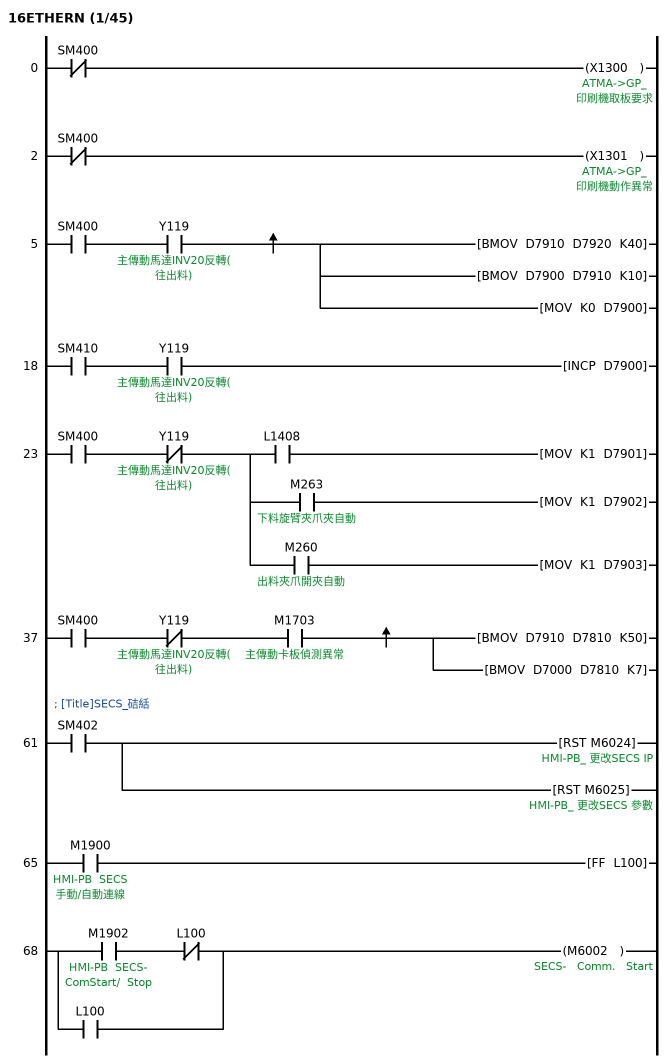
[picture p96: ladder of 16ETHERN, rungs at steps 0 to 68]
0     LDI     SM400
      OUT     X1300  ; ATMA->GP_印刷機取板要求
2     LDI     SM400
      OUT     X1301  ; ATMA->GP_印刷機動作異常
5     LD      SM400
      AND     Y119  ; 主傳動馬達INV20反轉(往出料)
      MEP
      BMOV    D7910 D7920 K40
      BMOV    D7900 D7910 K10
      MOV     K0 D7900
18    LD      SM410
      AND     Y119  ; 主傳動馬達INV20反轉(往出料)
      INCP    D7900
23    LD      SM400
      ANI     Y119  ; 主傳動馬達INV20反轉(往出料)
      MPS
      AND     L1408
      MOV     K1 D7901
      MRD
      AND     M263  ; 下料旋臂夾爪夾自動
      MOV     K1 D7902
      MPP
      AND     M260  ; 出料夾爪開夾自動
      MOV     K1 D7903
37    LD      SM400
      ANI     Y119  ; 主傳動馬達INV20反轉(往出料)
      AND     M1703  ; 主傳動卡板偵測異常
      MEP
      BMOV    D7910 D7810 K50
      BMOV    D7000 D7810 K7
; [Title]SECS_連線
61    LD      SM402
      RST     M6024  ; HMI-PB_ 更改SECS IP
      RST     M6025  ; HMI-PB_ 更改SECS 參數
65    LD      M1900  ; HMI-PB  SECS    手動/自動連線
      FF      L100
68    LD      M1902  ; HMI-PB  SECS-ComStart/  Stop
      ANI     L100
      OR      L100
      OUT     M6002  ; SECS-   Comm.   Start
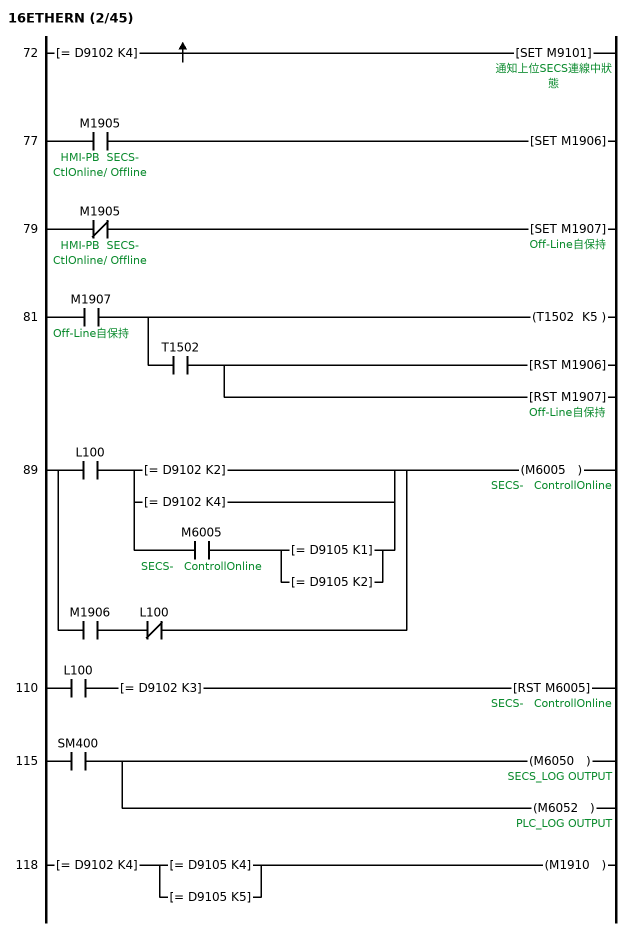
72    LD=     D9102 K4
      MEP
      SET     M9101  ; 通知上位SECS連線中狀態
77    LD      M1905  ; HMI-PB  SECS-CtlOnline/ Offline
      SET     M1906
79    LDI     M1905  ; HMI-PB  SECS-CtlOnline/ Offline
      SET     M1907  ; Off-Line自保持
81    LD      M1907  ; Off-Line自保持
      OUT     T1502 K5
      AND     T1502
      RST     M1906
      RST     M1907  ; Off-Line自保持
89    LD      L100
      LD=     D9102 K2
      OR=     D9102 K4
      LD      M6005  ; SECS-   ControllOnline
      LD=     D9105 K1
      OR=     D9105 K2
      ANB
      ORB
      ANB
      LD      M1906
      ANI     L100
      ORB
      OUT     M6005  ; SECS-   ControllOnline
110   LD      L100
      AND=    D9102 K3
      RST     M6005  ; SECS-   ControllOnline
115   LD      SM400
      OUT     M6050  ; SECS_LOG OUTPUT
      OUT     M6052  ; PLC_LOG OUTPUT
118   LD=     D9102 K4
      LD=     D9105 K4
      OR=     D9105 K5
      ANB
      OUT     M1910
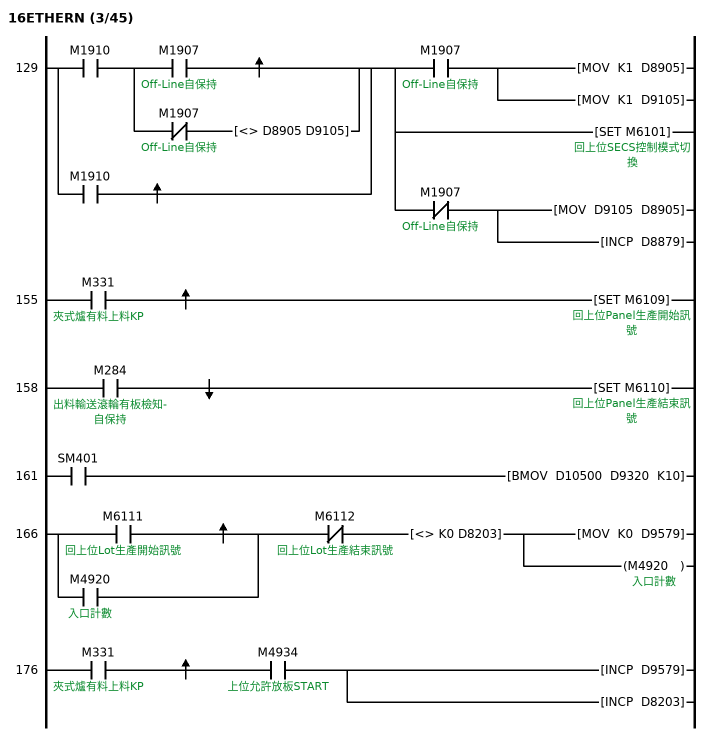
129   LD      M1910
      LD      M1907  ; Off-Line自保持
      MEP
      LDI     M1907  ; Off-Line自保持
      AND<>   D8905 D9105
      ORB
      ANB
      LD      M1910
      MEP
      ORB
      MPS
      AND     M1907  ; Off-Line自保持
      MOV     K1 D8905
      MOV     K1 D9105
      MPP
      SET     M6101  ; 回上位SECS控制模式切換
      ANI     M1907  ; Off-Line自保持
      MOV     D9105 D8905
      INCP    D8879
155   LD      M331  ; 夾式爐有料上料KP
      MEP
      SET     M6109  ; 回上位Panel生產開始訊號
158   LD      M284  ; 出料輸送滾輪有板檢知-自保持
      MEF
      SET     M6110  ; 回上位Panel生產結束訊號
161   LD      SM401
      BMOV    D10500 D9320 K10
166   LD      M6111  ; 回上位Lot生產開始訊號
      MEP
      OR      M4920  ; 入口計數
      ANI     M6112  ; 回上位Lot生產結束訊號
      AND<>   K0 D8203
      MOV     K0 D9579
      OUT     M4920  ; 入口計數
176   LD      M331  ; 夾式爐有料上料KP
      MEP
      AND     M4934  ; 上位允許放板START
      INCP    D9579
      INCP    D8203
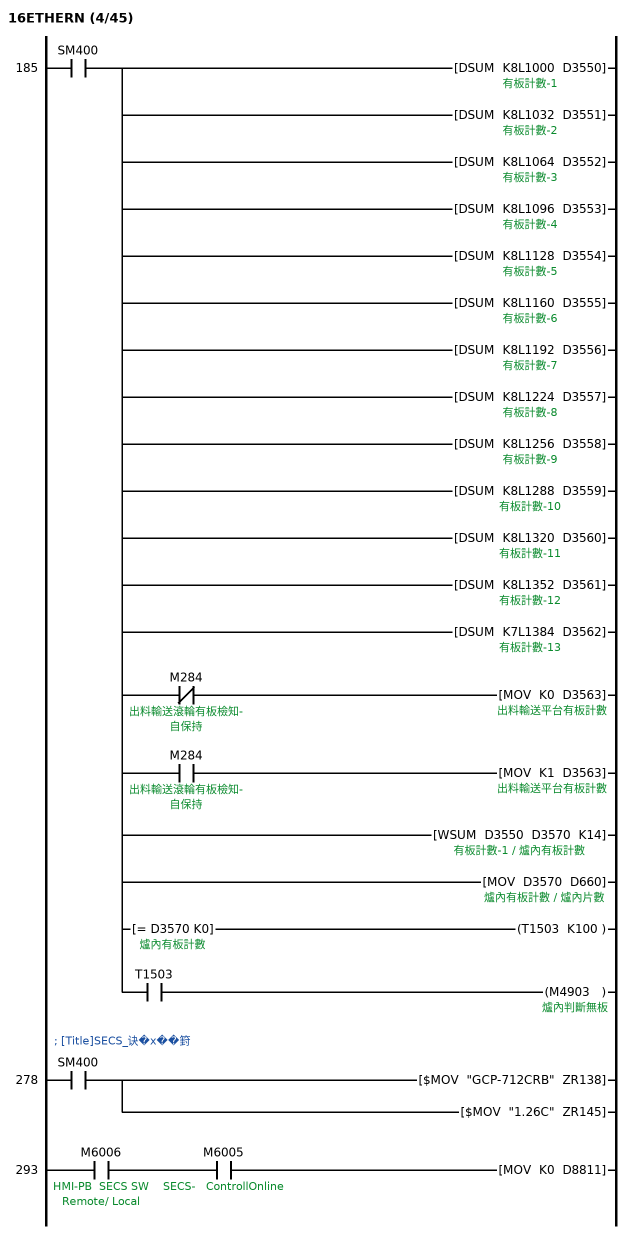
185   LD      SM400
      DSUM    K8L1000 D3550  ; 有板計數-1
      DSUM    K8L1032 D3551  ; 有板計數-2
      DSUM    K8L1064 D3552  ; 有板計數-3
      DSUM    K8L1096 D3553  ; 有板計數-4
      DSUM    K8L1128 D3554  ; 有板計數-5
      DSUM    K8L1160 D3555  ; 有板計數-6
      DSUM    K8L1192 D3556  ; 有板計數-7
      DSUM    K8L1224 D3557  ; 有板計數-8
      DSUM    K8L1256 D3558  ; 有板計數-9
      DSUM    K8L1288 D3559  ; 有板計數-10
      DSUM    K8L1320 D3560  ; 有板計數-11
      DSUM    K8L1352 D3561  ; 有板計數-12
      DSUM    K7L1384 D3562  ; 有板計數-13
      MPS
      ANI     M284  ; 出料輸送滾輪有板檢知-自保持
      MOV     K0 D3563  ; 出料輸送平台有板計數
      MRD
      AND     M284  ; 出料輸送滾輪有板檢知-自保持
      MOV     K1 D3563
      MPP
      WSUM    D3550 D3570 K14  ; 爐內有板計數
      MOV     D3570 D660  ; 爐內片數
      MPS
      AND=    D3570 K0  ; 爐內有板計數
      OUT     T1503 K100
      MPP
      AND     T1503
      OUT     M4903  ; 爐內判斷無板
; [Title]SECS_機台狀態
278   LD      SM400
      $MOV    "GCP-712CRB" ZR138
      $MOV    "1.26C" ZR145
293   LD      M6006  ; HMI-PB  SECS SW  Remote/ Local
      AND     M6005  ; SECS-   ControllOnline
      MOV     K0 D8811
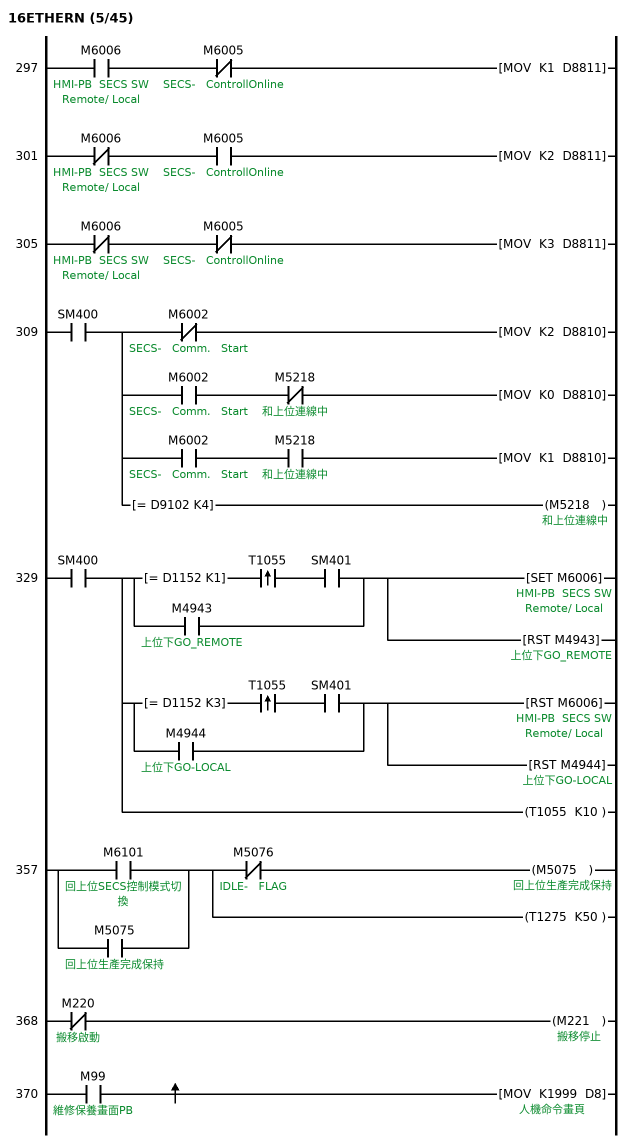
297   LD      M6006  ; HMI-PB  SECS SW  Remote/ Local
      ANI     M6005  ; SECS-   ControllOnline
      MOV     K1 D8811
301   LDI     M6006  ; HMI-PB  SECS SW  Remote/ Local
      AND     M6005  ; SECS-   ControllOnline
      MOV     K2 D8811
305   LDI     M6006  ; HMI-PB  SECS SW  Remote/ Local
      ANI     M6005  ; SECS-   ControllOnline
      MOV     K3 D8811
309   LD      SM400
      MPS
      ANI     M6002  ; SECS-   Comm.   Start
      MOV     K2 D8810
      MRD
      AND     M6002  ; SECS-   Comm.   Start
      ANI     M5218  ; 和上位連線中
      MOV     K0 D8810
      MRD
      AND     M6002  ; SECS-   Comm.   Start
      AND     M5218  ; 和上位連線中
      MOV     K1 D8810
      MPP
      AND=    D9102 K4
      OUT     M5218  ; 和上位連線中
329   LD      SM400
      MPS
      LD=     D1152 K1
      ANDP    T1055
      AND     SM401
      OR      M4943  ; 上位下GO_REMOTE
      ANB
      SET     M6006  ; HMI-PB  SECS SW  Remote/ Local
      RST     M4943  ; 上位下GO_REMOTE
      MRD
      LD=     D1152 K3
      ANDP    T1055
      AND     SM401
      OR      M4944  ; 上位下GO-LOCAL
      ANB
      RST     M6006  ; HMI-PB  SECS SW  Remote/ Local
      RST     M4944  ; 上位下GO-LOCAL
      MPP
      OUT     T1055 K10
357   LD      M6101  ; 回上位SECS控制模式切換
      OR      M5075  ; 回上位生產完成保持
      MPS
      ANI     M5076  ; IDLE-   FLAG
      OUT     M5075  ; 回上位生產完成保持
      MPP
      OUT     T1275 K50
368   LDI     M220  ; 搬移啟動
      OUT     M221  ; 搬移停止
370   LD      M99  ; 維修保養畫面PB
      MEP
      MOV     K1999 D8  ; 人機命令畫頁
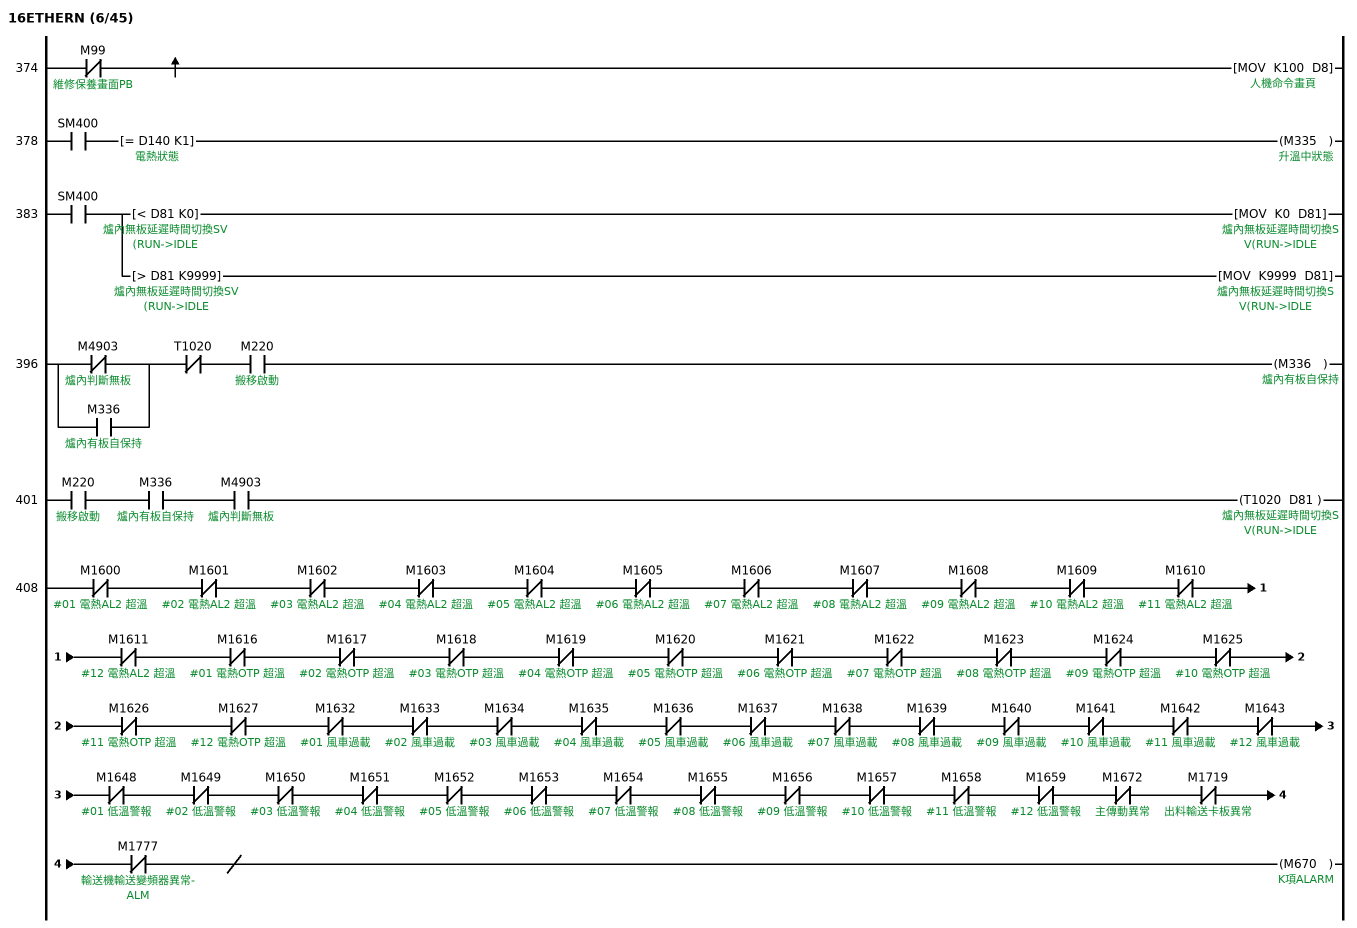
374   LDI     M99  ; 維修保養畫面PB
      MEP
      MOV     K100 D8
378   LD      SM400
      AND=    D140 K1  ; 電熱狀態
      OUT     M335  ; 升溫中狀態
383   LD      SM400
      MPS
      AND<    D81 K0  ; 爐內無板延遲時間切換SV(RUN->IDLE
      MOV     K0 D81
      MPP
      AND>    D81 K9999  ; 爐內無板延遲時間切換SV(RUN->IDLE
      MOV     K9999 D81
396   LDI     M4903  ; 爐內判斷無板
      OR      M336  ; 爐內有板自保持
      ANI     T1020
      AND     M220  ; 搬移啟動
      OUT     M336  ; 爐內有板自保持
401   LD      M220  ; 搬移啟動
      AND     M336  ; 爐內有板自保持
      AND     M4903  ; 爐內判斷無板
      OUT     T1020 D81  ; 爐內無板延遲時間切換SV(RUN->IDLE
408   LDI     M1600  ; #01 電熱AL2 超溫
      ANI     M1601  ; #02 電熱AL2 超溫
      ANI     M1602  ; #03 電熱AL2 超溫
      ANI     M1603  ; #04 電熱AL2 超溫
      ANI     M1604  ; #05 電熱AL2 超溫
      ANI     M1605  ; #06 電熱AL2 超溫
      ANI     M1606  ; #07 電熱AL2 超溫
      ANI     M1607  ; #08 電熱AL2 超溫
      ANI     M1608  ; #09 電熱AL2 超溫
      ANI     M1609  ; #10 電熱AL2 超溫
      ANI     M1610  ; #11 電熱AL2 超溫
      ANI     M1611  ; #12 電熱AL2 超溫
      ANI     M1616  ; #01 電熱OTP 超溫
      ANI     M1617  ; #02 電熱OTP 超溫
      ANI     M1618  ; #03 電熱OTP 超溫
      ANI     M1619  ; #04 電熱OTP 超溫
      ANI     M1620  ; #05 電熱OTP 超溫
      ANI     M1621  ; #06 電熱OTP 超溫
      ANI     M1622  ; #07 電熱OTP 超溫
      ANI     M1623  ; #08 電熱OTP 超溫
      ANI     M1624  ; #09 電熱OTP 超溫
      ANI     M1625  ; #10 電熱OTP 超溫
      ANI     M1626  ; #11 電熱OTP 超溫
      ANI     M1627  ; #12 電熱OTP 超溫
      ANI     M1632  ; #01 風車過載
      ANI     M1633  ; #02 風車過載
      ANI     M1634  ; #03 風車過載
      ANI     M1635  ; #04 風車過載
      ANI     M1636  ; #05 風車過載
      ANI     M1637  ; #06 風車過載
      ANI     M1638  ; #07 風車過載
      ANI     M1639  ; #08 風車過載
      ANI     M1640  ; #09 風車過載
      ANI     M1641  ; #10 風車過載
      ANI     M1642  ; #11 風車過載
      ANI     M1643  ; #12 風車過載
      ANI     M1648  ; #01 低溫警報
      ANI     M1649  ; #02 低溫警報
      ANI     M1650  ; #03 低溫警報
      ANI     M1651  ; #04 低溫警報
      ANI     M1652  ; #05 低溫警報
      ANI     M1653  ; #06 低溫警報
      ANI     M1654  ; #07 低溫警報
      ANI     M1655  ; #08 低溫警報
      ANI     M1656  ; #09 低溫警報
      ANI     M1657  ; #10 低溫警報
      ANI     M1658  ; #11 低溫警報
      ANI     M1659  ; #12 低溫警報
      ANI     M1672  ; 主傳動異常
      ANI     M1719  ; 出料輸送卡板異常
      ANI     M1777  ; 輸送機輸送變頻器異常-ALM
      INV
      OUT     M670  ; K項ALARM
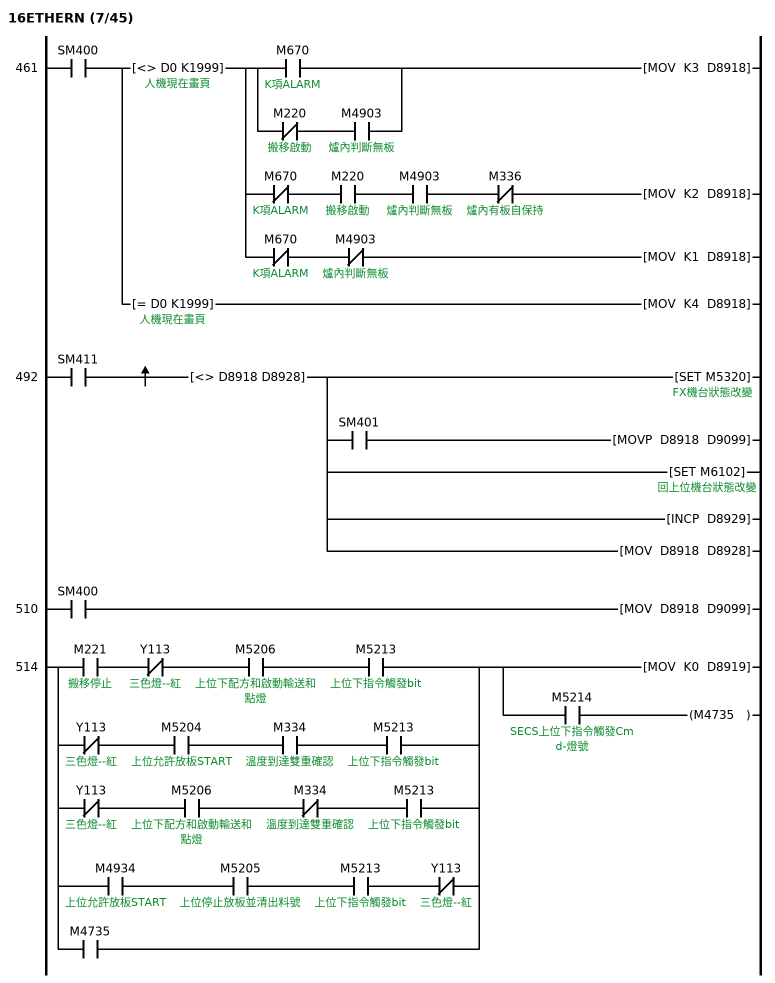
461   LD      SM400
      MPS
      AND<>   D0 K1999  ; 人機現在畫頁
      MPS
      LD      M670  ; K項ALARM
      LDI     M220  ; 搬移啟動
      AND     M4903  ; 爐內判斷無板
      ORB
      ANB
      MOV     K3 D8918
      MRD
      ANI     M670  ; K項ALARM
      AND     M220  ; 搬移啟動
      AND     M4903  ; 爐內判斷無板
      ANI     M336  ; 爐內有板自保持
      MOV     K2 D8918
      MPP
      ANI     M670  ; K項ALARM
      ANI     M4903  ; 爐內判斷無板
      MOV     K1 D8918
      MPP
      AND=    D0 K1999  ; 人機現在畫頁
      MOV     K4 D8918
492   LD      SM411
      MEP
      AND<>   D8918 D8928
      SET     M5320  ; FX機台狀態改變
      MPS
      AND     SM401
      MOVP    D8918 D9099
      MPP
      SET     M6102  ; 回上位機台狀態改變
      INCP    D8929
      MOV     D8918 D8928
510   LD      SM400
      MOV     D8918 D9099
514   LD      M221  ; 搬移停止
      ANI     Y113  ; 三色燈--紅
      AND     M5206  ; 上位下配方和啟動輸送和點燈
      AND     M5213  ; 上位下指令觸發bit
      LDI     Y113  ; 三色燈--紅
      AND     M5204  ; 上位允許放板START
      AND     M334  ; 溫度到達雙重確認
      AND     M5213  ; 上位下指令觸發bit
      ORB
      LDI     Y113  ; 三色燈--紅
      AND     M5206  ; 上位下配方和啟動輸送和點燈
      ANI     M334  ; 溫度到達雙重確認
      AND     M5213  ; 上位下指令觸發bit
      ORB
      LD      M4934  ; 上位允許放板START
      AND     M5205  ; 上位停止放板並清出料號
      AND     M5213  ; 上位下指令觸發bit
      ANI     Y113  ; 三色燈--紅
      ORB
      OR      M4735
      MOV     K0 D8919
      AND     M5214  ; SECS上位下指令觸發Cmd-燈號
      OUT     M4735
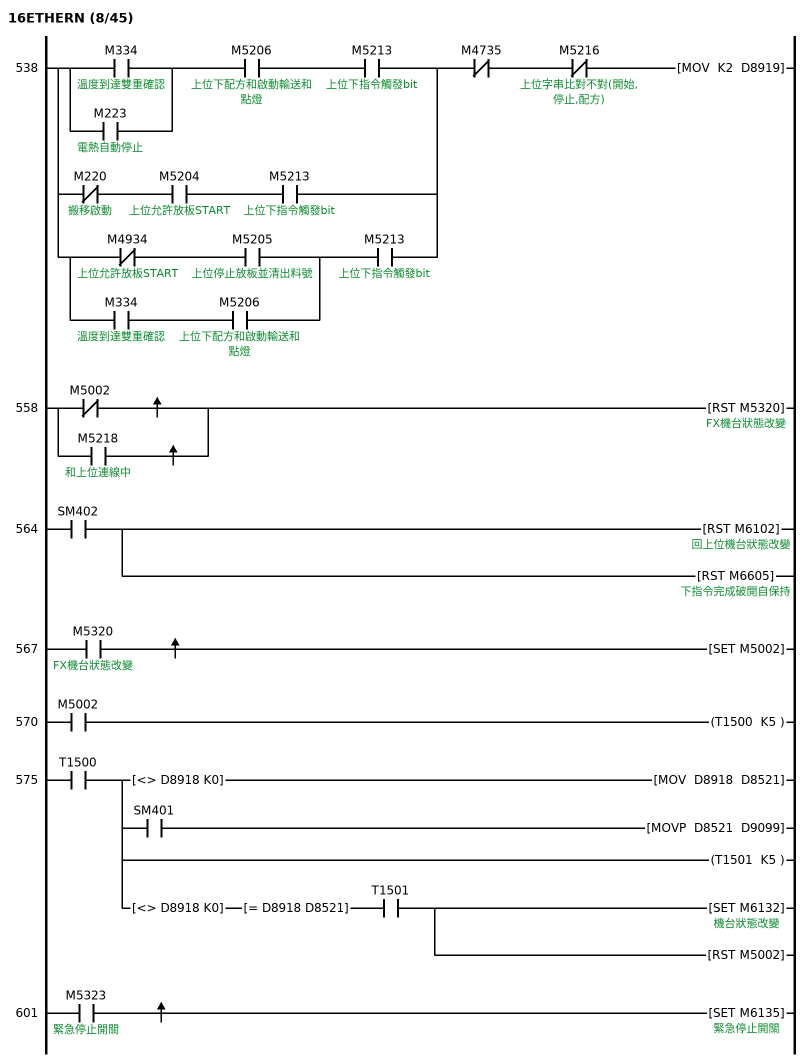
538   LD      M334  ; 溫度到達雙重確認
      OR      M223  ; 電熱自動停止
      AND     M5206  ; 上位下配方和啟動輸送和點燈
      AND     M5213  ; 上位下指令觸發bit
      LDI     M220  ; 搬移啟動
      AND     M5204  ; 上位允許放板START
      AND     M5213  ; 上位下指令觸發bit
      ORB
      LDI     M4934  ; 上位允許放板START
      AND     M5205  ; 上位停止放板並清出料號
      LD      M334  ; 溫度到達雙重確認
      AND     M5206  ; 上位下配方和啟動輸送和點燈
      ORB
      AND     M5213  ; 上位下指令觸發bit
      ORB
      ANI     M4735
      ANI     M5216  ; 上位字串比對不對(開始,停止,配方)
      MOV     K2 D8919
558   LDI     M5002
      MEP
      LD      M5218  ; 和上位連線中
      MEP
      ORB
      RST     M5320  ; FX機台狀態改變
564   LD      SM402
      RST     M6102  ; 回上位機台狀態改變
      RST     M6605  ; 下指令完成破開自保持
567   LD      M5320  ; FX機台狀態改變
      MEP
      SET     M5002
570   LD      M5002
      OUT     T1500 K5
575   LD      T1500
      MPS
      AND<>   D8918 K0
      MOV     D8918 D8521
      MRD
      AND     SM401
      MOVP    D8521 D9099
      MPP
      OUT     T1501 K5
      AND<>   D8918 K0
      AND=    D8918 D8521
      AND     T1501
      SET     M6132  ; 機台狀態改變
      RST     M5002
601   LD      M5323  ; 緊急停止開關
      MEP
      SET     M6135  ; 緊急停止開關
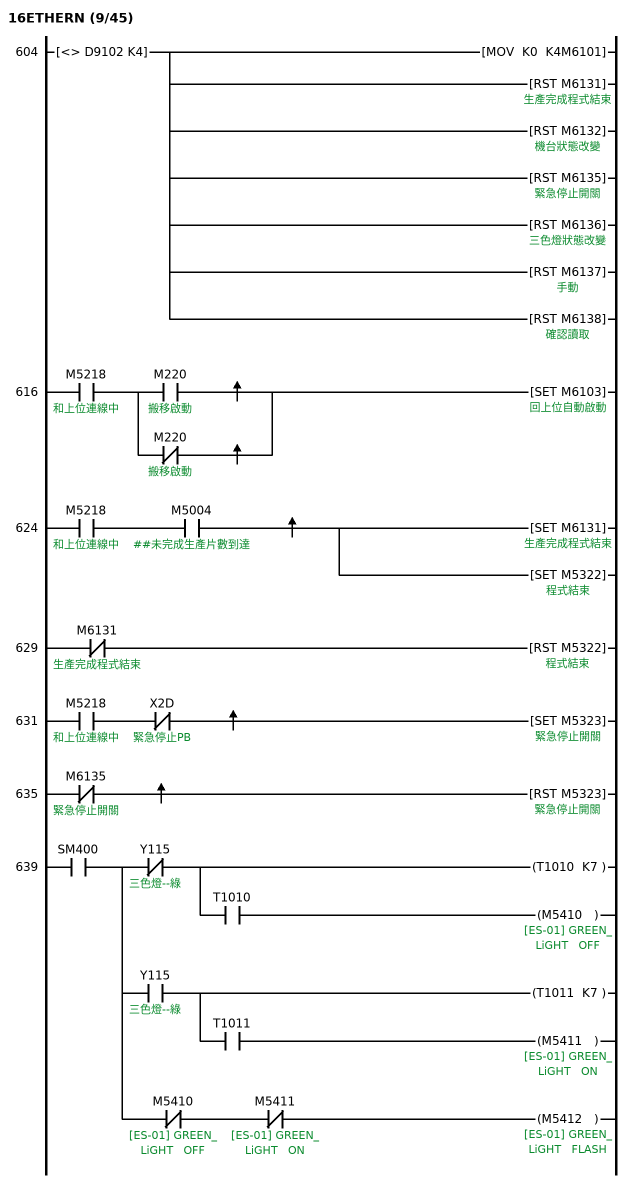
604   LD<>    D9102 K4
      MOV     K0 K4M6101
      RST     M6131  ; 生產完成程式結束
      RST     M6132  ; 機台狀態改變
      RST     M6135  ; 緊急停止開關
      RST     M6136  ; 三色燈狀態改變
      RST     M6137  ; 手動
      RST     M6138  ; 確認讀取
616   LD      M5218  ; 和上位連線中
      LD      M220  ; 搬移啟動
      MEP
      LDI     M220  ; 搬移啟動
      MEP
      ORB
      ANB
      SET     M6103  ; 回上位自動啟動
624   LD      M5218  ; 和上位連線中
      AND     M5004  ; ##未完成生產片數到達
      MEP
      SET     M6131  ; 生產完成程式結束
      SET     M5322  ; 程式結束
629   LDI     M6131  ; 生產完成程式結束
      RST     M5322  ; 程式結束
631   LD      M5218  ; 和上位連線中
      ANI     X2D  ; 緊急停止PB
      MEP
      SET     M5323  ; 緊急停止開關
635   LDI     M6135  ; 緊急停止開關
      MEP
      RST     M5323  ; 緊急停止開關
639   LD      SM400
      MPS
      ANI     Y115  ; 三色燈--綠
      OUT     T1010 K7
      AND     T1010
      OUT     M5410  ; [ES-01] GREEN_  LiGHT   OFF
      MRD
      AND     Y115  ; 三色燈--綠
      OUT     T1011 K7
      AND     T1011
      OUT     M5411  ; [ES-01] GREEN_  LiGHT   ON
      MPP
      ANI     M5410  ; [ES-01] GREEN_  LiGHT   OFF
      ANI     M5411  ; [ES-01] GREEN_  LiGHT   ON
      OUT     M5412  ; [ES-01] GREEN_  LiGHT   FLASH
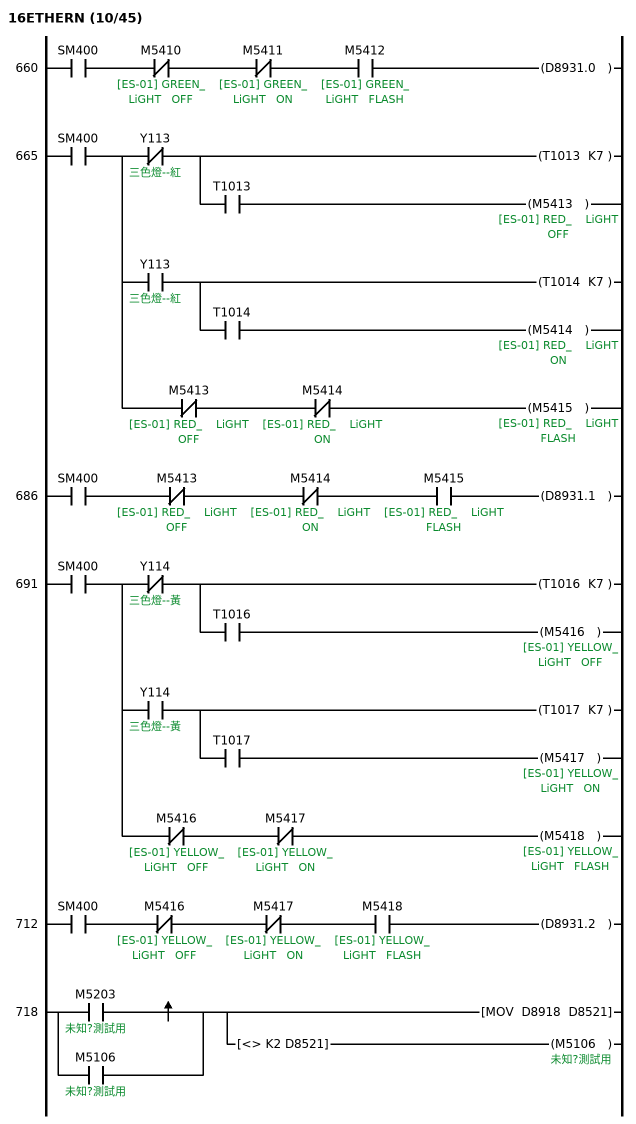
660   LD      SM400
      ANI     M5410  ; [ES-01] GREEN_  LiGHT   OFF
      ANI     M5411  ; [ES-01] GREEN_  LiGHT   ON
      AND     M5412  ; [ES-01] GREEN_  LiGHT   FLASH
      OUT     D8931.0
665   LD      SM400
      MPS
      ANI     Y113  ; 三色燈--紅
      OUT     T1013 K7
      AND     T1013
      OUT     M5413  ; [ES-01] RED_    LiGHT   OFF
      MRD
      AND     Y113  ; 三色燈--紅
      OUT     T1014 K7
      AND     T1014
      OUT     M5414  ; [ES-01] RED_    LiGHT   ON
      MPP
      ANI     M5413  ; [ES-01] RED_    LiGHT   OFF
      ANI     M5414  ; [ES-01] RED_    LiGHT   ON
      OUT     M5415  ; [ES-01] RED_    LiGHT   FLASH
686   LD      SM400
      ANI     M5413  ; [ES-01] RED_    LiGHT   OFF
      ANI     M5414  ; [ES-01] RED_    LiGHT   ON
      AND     M5415  ; [ES-01] RED_    LiGHT   FLASH
      OUT     D8931.1
691   LD      SM400
      MPS
      ANI     Y114  ; 三色燈--黃
      OUT     T1016 K7
      AND     T1016
      OUT     M5416  ; [ES-01] YELLOW_ LiGHT   OFF
      MRD
      AND     Y114  ; 三色燈--黃
      OUT     T1017 K7
      AND     T1017
      OUT     M5417  ; [ES-01] YELLOW_ LiGHT   ON
      MPP
      ANI     M5416  ; [ES-01] YELLOW_ LiGHT   OFF
      ANI     M5417  ; [ES-01] YELLOW_ LiGHT   ON
      OUT     M5418  ; [ES-01] YELLOW_ LiGHT   FLASH
712   LD      SM400
      ANI     M5416  ; [ES-01] YELLOW_ LiGHT   OFF
      ANI     M5417  ; [ES-01] YELLOW_ LiGHT   ON
      AND     M5418  ; [ES-01] YELLOW_ LiGHT   FLASH
      OUT     D8931.2
718   LD      M5203  ; 未知?測試用
      MEP
      OR      M5106  ; 未知?測試用
      MOV     D8918 D8521
      AND<>   K2 D8521
      OUT     M5106  ; 未知?測試用
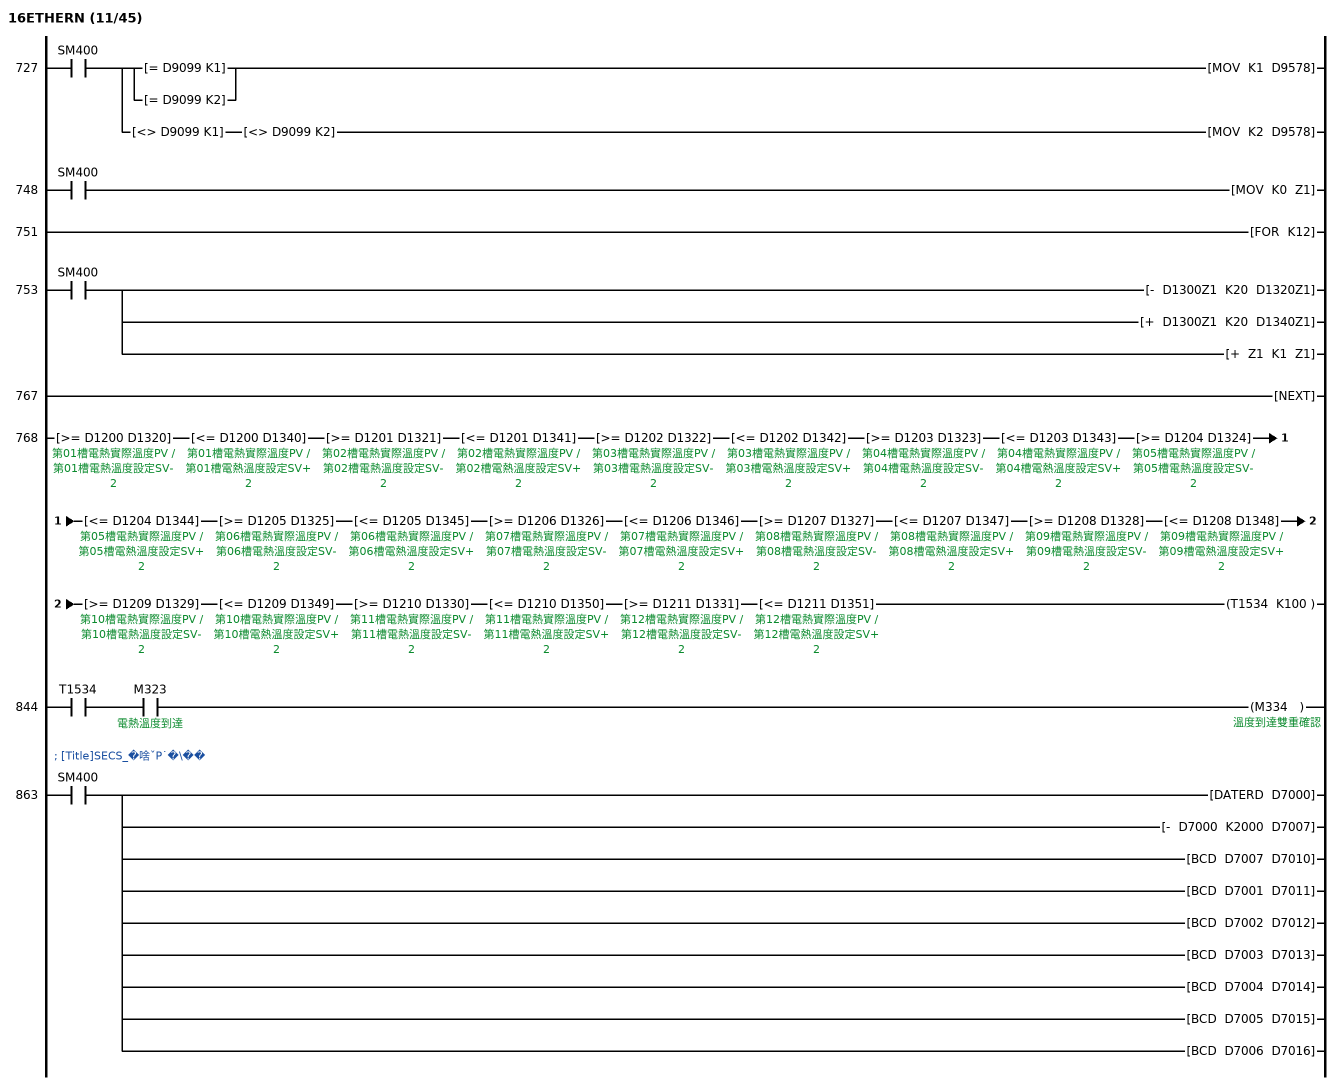
727   LD      SM400
      MPS
      LD=     D9099 K1
      OR=     D9099 K2
      ANB
      MOV     K1 D9578
      MPP
      AND<>   D9099 K1
      AND<>   D9099 K2
      MOV     K2 D9578
748   LD      SM400
      MOV     K0 Z1
751   FOR     K12
753   LD      SM400
      -       D1300Z1 K20 D1320Z1
      +       D1300Z1 K20 D1340Z1
      +       Z1 K1 Z1
767   NEXT
768   LD>=    D1200 D1320  ; 第01槽電熱實際溫度PV / 第01槽電熱溫度設定SV-2
      AND<=   D1200 D1340  ; 第01槽電熱實際溫度PV / 第01槽電熱溫度設定SV+2
      AND>=   D1201 D1321  ; 第02槽電熱實際溫度PV / 第02槽電熱溫度設定SV-2
      AND<=   D1201 D1341  ; 第02槽電熱實際溫度PV / 第02槽電熱溫度設定SV+2
      AND>=   D1202 D1322  ; 第03槽電熱實際溫度PV / 第03槽電熱溫度設定SV-2
      AND<=   D1202 D1342  ; 第03槽電熱實際溫度PV / 第03槽電熱溫度設定SV+2
      AND>=   D1203 D1323  ; 第04槽電熱實際溫度PV / 第04槽電熱溫度設定SV-2
      AND<=   D1203 D1343  ; 第04槽電熱實際溫度PV / 第04槽電熱溫度設定SV+2
      AND>=   D1204 D1324  ; 第05槽電熱實際溫度PV / 第05槽電熱溫度設定SV-2
      AND<=   D1204 D1344  ; 第05槽電熱實際溫度PV / 第05槽電熱溫度設定SV+2
      AND>=   D1205 D1325  ; 第06槽電熱實際溫度PV / 第06槽電熱溫度設定SV-2
      AND<=   D1205 D1345  ; 第06槽電熱實際溫度PV / 第06槽電熱溫度設定SV+2
      AND>=   D1206 D1326  ; 第07槽電熱實際溫度PV / 第07槽電熱溫度設定SV-2
      AND<=   D1206 D1346  ; 第07槽電熱實際溫度PV / 第07槽電熱溫度設定SV+2
      AND>=   D1207 D1327  ; 第08槽電熱實際溫度PV / 第08槽電熱溫度設定SV-2
      AND<=   D1207 D1347  ; 第08槽電熱實際溫度PV / 第08槽電熱溫度設定SV+2
      AND>=   D1208 D1328  ; 第09槽電熱實際溫度PV / 第09槽電熱溫度設定SV-2
      AND<=   D1208 D1348  ; 第09槽電熱實際溫度PV / 第09槽電熱溫度設定SV+2
      AND>=   D1209 D1329  ; 第10槽電熱實際溫度PV / 第10槽電熱溫度設定SV-2
      AND<=   D1209 D1349  ; 第10槽電熱實際溫度PV / 第10槽電熱溫度設定SV+2
      AND>=   D1210 D1330  ; 第11槽電熱實際溫度PV / 第11槽電熱溫度設定SV-2
      AND<=   D1210 D1350  ; 第11槽電熱實際溫度PV / 第11槽電熱溫度設定SV+2
      AND>=   D1211 D1331  ; 第12槽電熱實際溫度PV / 第12槽電熱溫度設定SV-2
      AND<=   D1211 D1351  ; 第12槽電熱實際溫度PV / 第12槽電熱溫度設定SV+2
      OUT     T1534 K100
844   LD      T1534
      AND     M323  ; 電熱溫度到達
      OUT     M334  ; 溫度到達雙重確認
; [Title]SECS_時間同步功能
863   LD      SM400
      DATERD  D7000
      -       D7000 K2000 D7007
      BCD     D7007 D7010
      BCD     D7001 D7011
      BCD     D7002 D7012
      BCD     D7003 D7013
      BCD     D7004 D7014
      BCD     D7005 D7015
      BCD     D7006 D7016
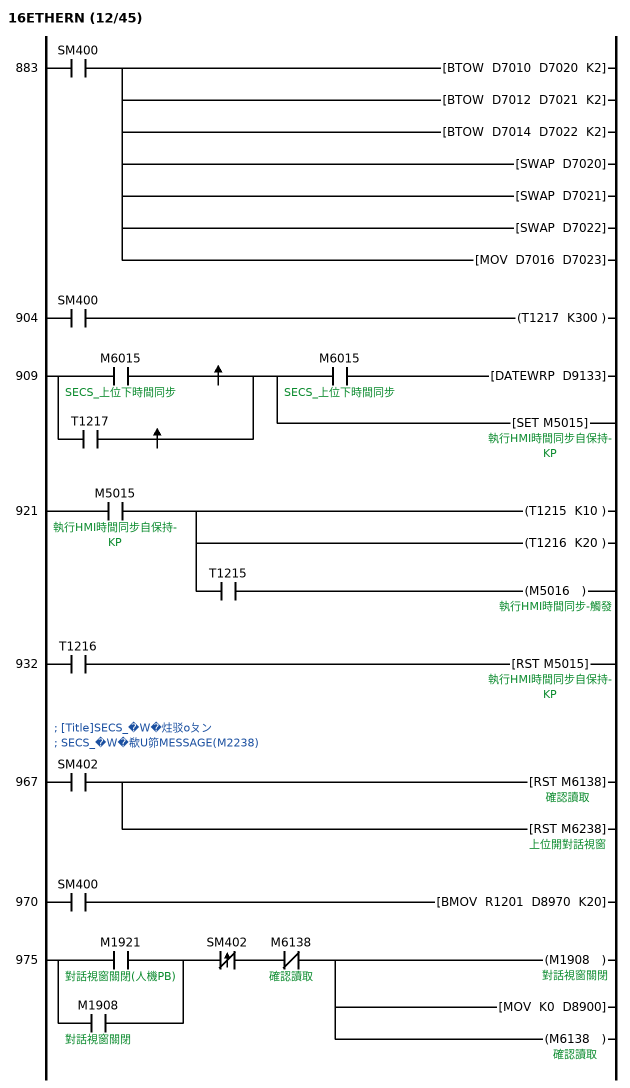
883   LD      SM400
      BTOW    D7010 D7020 K2
      BTOW    D7012 D7021 K2
      BTOW    D7014 D7022 K2
      SWAP    D7020
      SWAP    D7021
      SWAP    D7022
      MOV     D7016 D7023
904   LD      SM400
      OUT     T1217 K300
909   LD      M6015  ; SECS_上位下時間同步
      MEP
      LD      T1217
      MEP
      ORB
      MPS
      AND     M6015  ; SECS_上位下時間同步
      DATEWRP D9133
      MPP
      SET     M5015  ; 執行HMI時間同步自保持-KP
921   LD      M5015  ; 執行HMI時間同步自保持-KP
      OUT     T1215 K10
      OUT     T1216 K20
      AND     T1215
      OUT     M5016  ; 執行HMI時間同步-觸發
932   LD      T1216
      RST     M5015  ; 執行HMI時間同步自保持-KP
; [Title]SECS_上位觸發事件
; SECS_上位下達MESSAGE(M2238)
967   LD      SM402
      RST     M6138  ; 確認讀取
      RST     M6238  ; 上位開對話視窗
970   LD      SM400
      BMOV    R1201 D8970 K20
975   LD      M1921  ; 對話視窗關閉(人機PB)
      OR      M1908  ; 對話視窗關閉
      ANDPI   SM402
      ANI     M6138  ; 確認讀取
      OUT     M1908  ; 對話視窗關閉
      MOV     K0 D8900
      OUT     M6138  ; 確認讀取
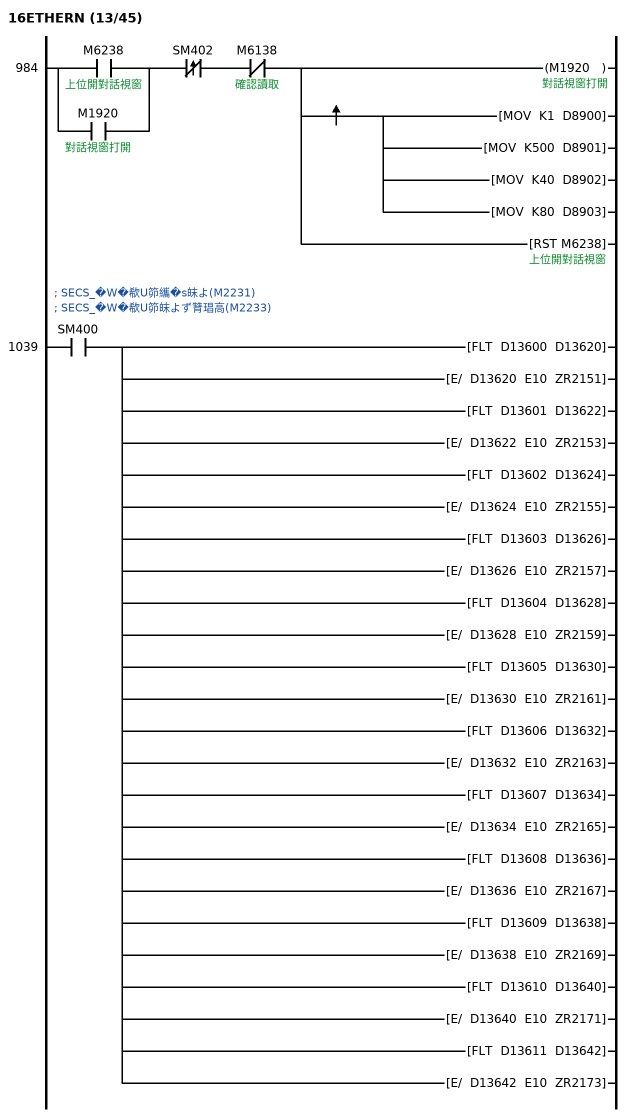
984   LD      M6238  ; 上位開對話視窗
      OR      M1920  ; 對話視窗打開
      ANDPI   SM402
      ANI     M6138  ; 確認讀取
      OUT     M1920  ; 對話視窗打開
      MPS
      MEP
      MOV     K1 D8900
      MOV     K500 D8901
      MOV     K40 D8902
      MOV     K80 D8903
      MPP
      RST     M6238  ; 上位開對話視窗
; SECS_上位下達儲存配方(M2231)
; SECS_上位下達配方內容查詢(M2233)
1039  LD      SM400
      FLT     D13600 D13620
      E/      D13620 E10 ZR2151
      FLT     D13601 D13622
      E/      D13622 E10 ZR2153
      FLT     D13602 D13624
      E/      D13624 E10 ZR2155
      FLT     D13603 D13626
      E/      D13626 E10 ZR2157
      FLT     D13604 D13628
      E/      D13628 E10 ZR2159
      FLT     D13605 D13630
      E/      D13630 E10 ZR2161
      FLT     D13606 D13632
      E/      D13632 E10 ZR2163
      FLT     D13607 D13634
      E/      D13634 E10 ZR2165
      FLT     D13608 D13636
      E/      D13636 E10 ZR2167
      FLT     D13609 D13638
      E/      D13638 E10 ZR2169
      FLT     D13610 D13640
      E/      D13640 E10 ZR2171
      FLT     D13611 D13642
      E/      D13642 E10 ZR2173
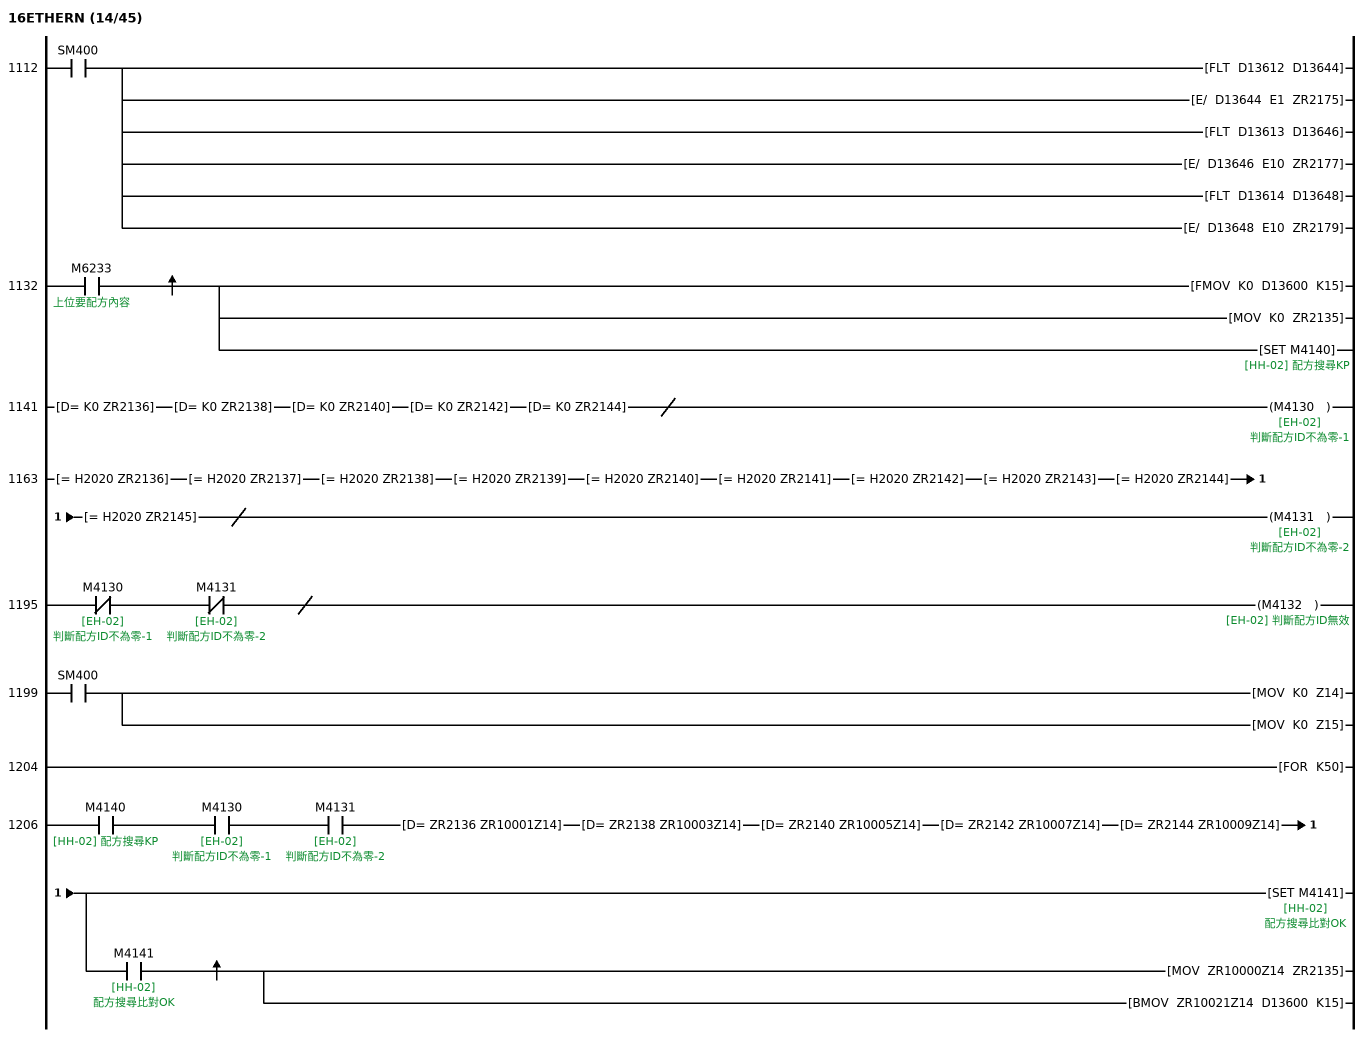
1112  LD      SM400
      FLT     D13612 D13644
      E/      D13644 E1 ZR2175
      FLT     D13613 D13646
      E/      D13646 E10 ZR2177
      FLT     D13614 D13648
      E/      D13648 E10 ZR2179
1132  LD      M6233  ; 上位要配方內容
      MEP
      FMOV    K0 D13600 K15
      MOV     K0 ZR2135
      SET     M4140  ; [HH-02] 配方搜尋KP
1141  LDD=    K0 ZR2136
      ANDD=   K0 ZR2138
      ANDD=   K0 ZR2140
      ANDD=   K0 ZR2142
      ANDD=   K0 ZR2144
      INV
      OUT     M4130  ; [EH-02] 判斷配方ID不為零-1
1163  LD=     H2020 ZR2136
      AND=    H2020 ZR2137
      AND=    H2020 ZR2138
      AND=    H2020 ZR2139
      AND=    H2020 ZR2140
      AND=    H2020 ZR2141
      AND=    H2020 ZR2142
      AND=    H2020 ZR2143
      AND=    H2020 ZR2144
      AND=    H2020 ZR2145
      INV
      OUT     M4131  ; [EH-02] 判斷配方ID不為零-2
1195  LDI     M4130  ; [EH-02] 判斷配方ID不為零-1
      ANI     M4131  ; [EH-02] 判斷配方ID不為零-2
      INV
      OUT     M4132  ; [EH-02] 判斷配方ID無效
1199  LD      SM400
      MOV     K0 Z14
      MOV     K0 Z15
1204  FOR     K50
1206  LD      M4140  ; [HH-02] 配方搜尋KP
      AND     M4130  ; [EH-02] 判斷配方ID不為零-1
      AND     M4131  ; [EH-02] 判斷配方ID不為零-2
      ANDD=   ZR2136 ZR10001Z14
      ANDD=   ZR2138 ZR10003Z14
      ANDD=   ZR2140 ZR10005Z14
      ANDD=   ZR2142 ZR10007Z14
      ANDD=   ZR2144 ZR10009Z14
      SET     M4141  ; [HH-02] 配方搜尋比對OK
      AND     M4141  ; [HH-02] 配方搜尋比對OK
      MEP
      MOV     ZR10000Z14 ZR2135
      BMOV    ZR10021Z14 D13600 K15
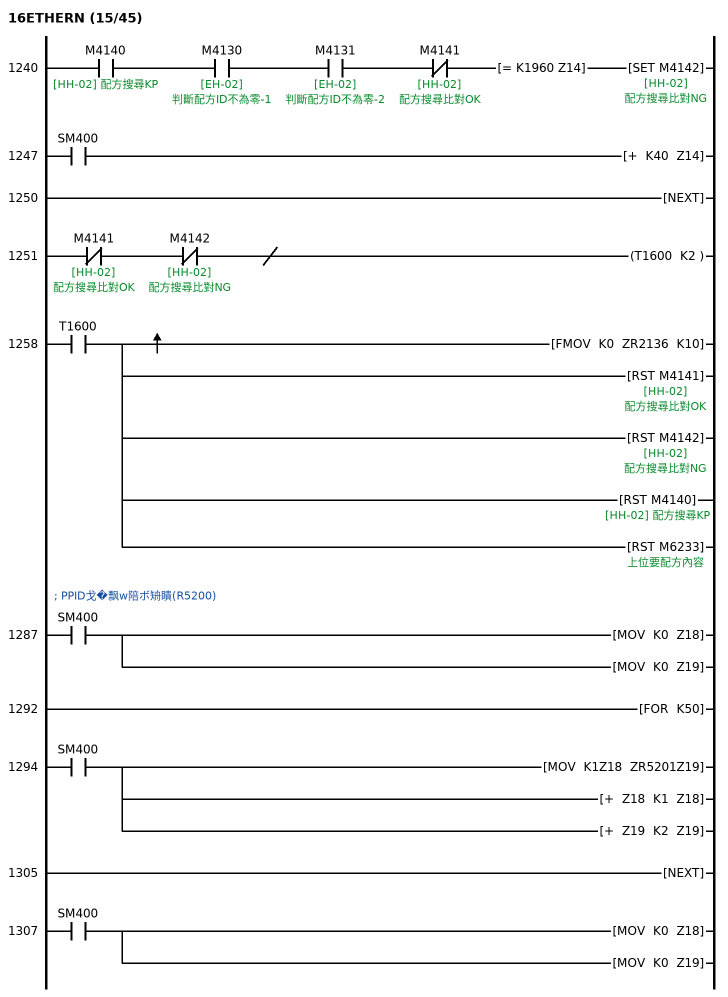
1240  LD      M4140  ; [HH-02] 配方搜尋KP
      AND     M4130  ; [EH-02] 判斷配方ID不為零-1
      AND     M4131  ; [EH-02] 判斷配方ID不為零-2
      ANI     M4141  ; [HH-02] 配方搜尋比對OK
      AND=    K1960 Z14
      SET     M4142  ; [HH-02] 配方搜尋比對NG
1247  LD      SM400
      +       K40 Z14
1250  NEXT
1251  LDI     M4141  ; [HH-02] 配方搜尋比對OK
      ANI     M4142  ; [HH-02] 配方搜尋比對NG
      INV
      OUT     T1600 K2
1258  LD      T1600
      MPS
      MEP
      FMOV    K0 ZR2136 K10
      MPP
      RST     M4141  ; [HH-02] 配方搜尋比對OK
      RST     M4142  ; [HH-02] 配方搜尋比對NG
      RST     M4140  ; [HH-02] 配方搜尋KP
      RST     M6233  ; 上位要配方內容
; PPID資料庫顯示處理(R5200)
1287  LD      SM400
      MOV     K0 Z18
      MOV     K0 Z19
1292  FOR     K50
1294  LD      SM400
      MOV     K1Z18 ZR5201Z19
      +       Z18 K1 Z18
      +       Z19 K2 Z19
1305  NEXT
1307  LD      SM400
      MOV     K0 Z18
      MOV     K0 Z19
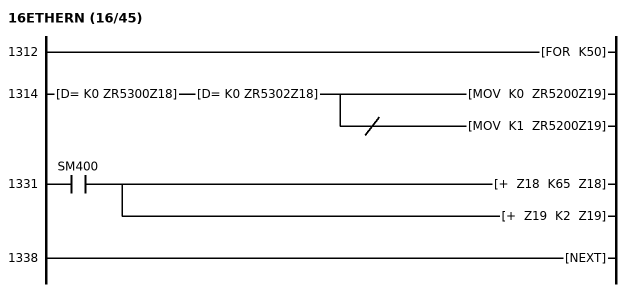
1312  FOR     K50
1314  LDD=    K0 ZR5300Z18
      ANDD=   K0 ZR5302Z18
      MOV     K0 ZR5200Z19
      INV
      MOV     K1 ZR5200Z19
1331  LD      SM400
      +       Z18 K65 Z18
      +       Z19 K2 Z19
1338  NEXT
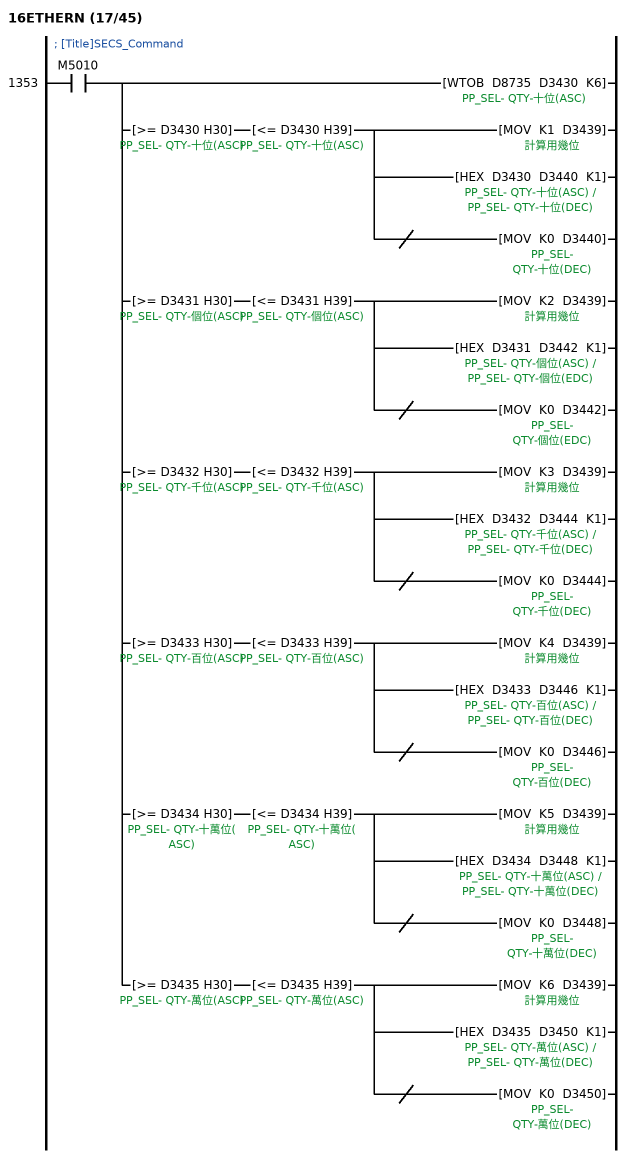
; [Title]SECS_Command
1353  LD      M5010
      WTOB    D8735 D3430 K6  ; PP_SEL- QTY-十位(ASC)
      MPS
      AND>=   D3430 H30  ; PP_SEL- QTY-十位(ASC)
      AND<=   D3430 H39  ; PP_SEL- QTY-十位(ASC)
      MOV     K1 D3439  ; 計算用幾位
      HEX     D3430 D3440 K1  ; PP_SEL- QTY-十位(DEC)
      INV
      MOV     K0 D3440
      MRD
      AND>=   D3431 H30  ; PP_SEL- QTY-個位(ASC)
      AND<=   D3431 H39  ; PP_SEL- QTY-個位(ASC)
      MOV     K2 D3439
      HEX     D3431 D3442 K1  ; PP_SEL- QTY-個位(EDC)
      INV
      MOV     K0 D3442
      MRD
      AND>=   D3432 H30  ; PP_SEL- QTY-千位(ASC)
      AND<=   D3432 H39  ; PP_SEL- QTY-千位(ASC)
      MOV     K3 D3439
      HEX     D3432 D3444 K1  ; PP_SEL- QTY-千位(DEC)
      INV
      MOV     K0 D3444
      MRD
      AND>=   D3433 H30  ; PP_SEL- QTY-百位(ASC)
      AND<=   D3433 H39  ; PP_SEL- QTY-百位(ASC)
      MOV     K4 D3439
      HEX     D3433 D3446 K1  ; PP_SEL- QTY-百位(DEC)
      INV
      MOV     K0 D3446
      MRD
      AND>=   D3434 H30  ; PP_SEL- QTY-十萬位(ASC)
      AND<=   D3434 H39  ; PP_SEL- QTY-十萬位(ASC)
      MOV     K5 D3439
      HEX     D3434 D3448 K1  ; PP_SEL- QTY-十萬位(DEC)
      INV
      MOV     K0 D3448
      MPP
      AND>=   D3435 H30  ; PP_SEL- QTY-萬位(ASC)
      AND<=   D3435 H39  ; PP_SEL- QTY-萬位(ASC)
      MOV     K6 D3439
      HEX     D3435 D3450 K1  ; PP_SEL- QTY-萬位(DEC)
      INV
      MOV     K0 D3450
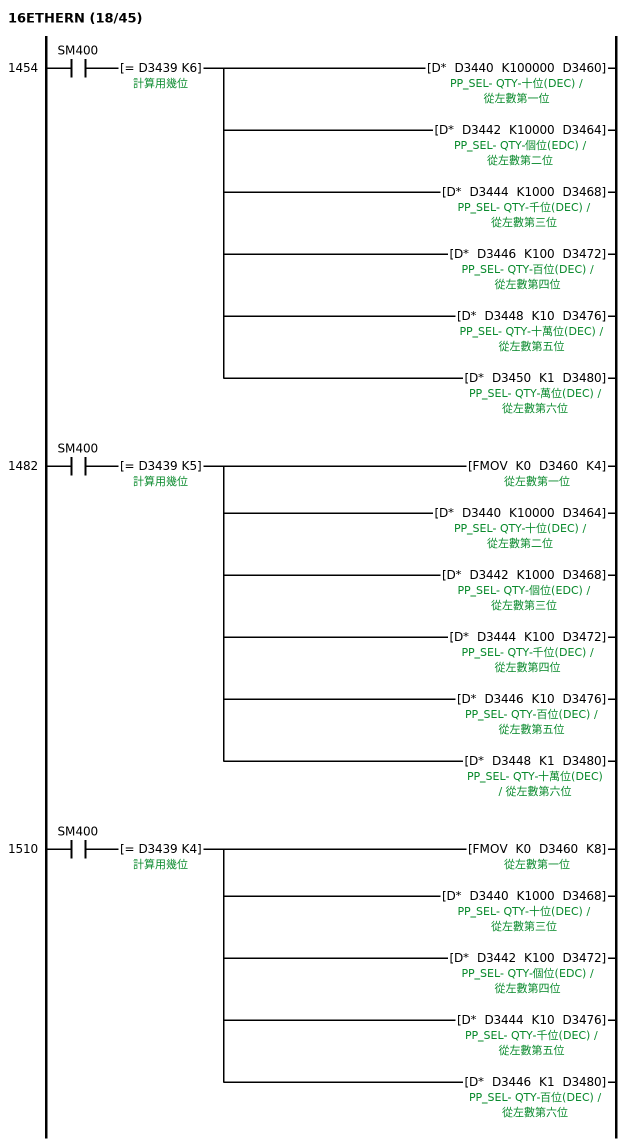
1454  LD      SM400
      AND=    D3439 K6  ; 計算用幾位
      D*      D3440 K100000 D3460  ; 從左數第一位
      D*      D3442 K10000 D3464  ; 從左數第二位
      D*      D3444 K1000 D3468  ; 從左數第三位
      D*      D3446 K100 D3472  ; 從左數第四位
      D*      D3448 K10 D3476  ; 從左數第五位
      D*      D3450 K1 D3480  ; 從左數第六位
1482  LD      SM400
      AND=    D3439 K5  ; 計算用幾位
      FMOV    K0 D3460 K4
      D*      D3440 K10000 D3464
      D*      D3442 K1000 D3468
      D*      D3444 K100 D3472
      D*      D3446 K10 D3476
      D*      D3448 K1 D3480
1510  LD      SM400
      AND=    D3439 K4  ; 計算用幾位
      FMOV    K0 D3460 K8
      D*      D3440 K1000 D3468
      D*      D3442 K100 D3472
      D*      D3444 K10 D3476
      D*      D3446 K1 D3480
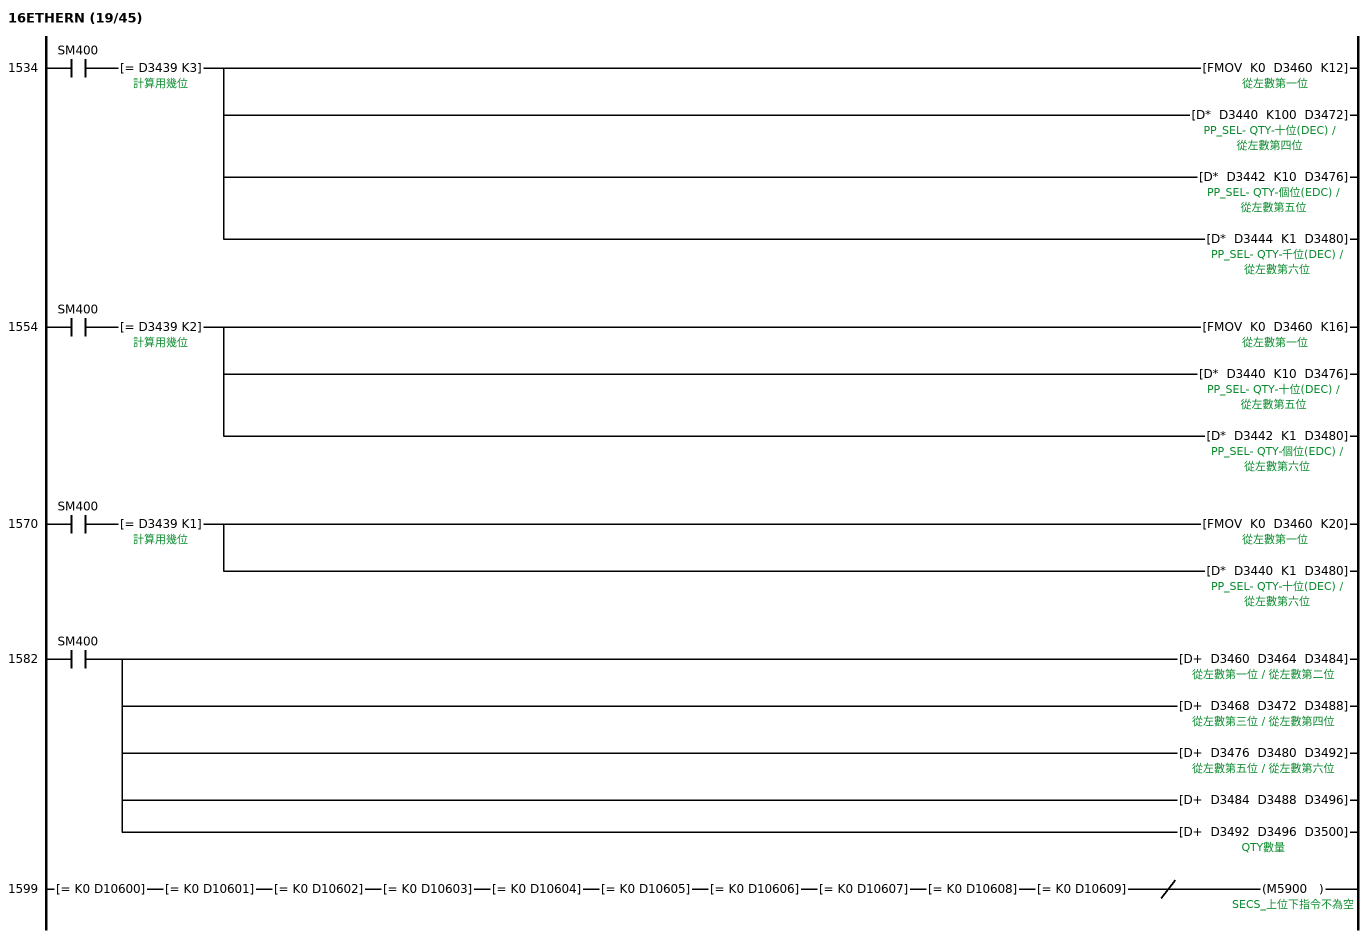
1534  LD      SM400
      AND=    D3439 K3  ; 計算用幾位
      FMOV    K0 D3460 K12
      D*      D3440 K100 D3472
      D*      D3442 K10 D3476
      D*      D3444 K1 D3480
1554  LD      SM400
      AND=    D3439 K2  ; 計算用幾位
      FMOV    K0 D3460 K16
      D*      D3440 K10 D3476
      D*      D3442 K1 D3480
1570  LD      SM400
      AND=    D3439 K1  ; 計算用幾位
      FMOV    K0 D3460 K20
      D*      D3440 K1 D3480
1582  LD      SM400
      D+      D3460 D3464 D3484
      D+      D3468 D3472 D3488
      D+      D3476 D3480 D3492
      D+      D3484 D3488 D3496
      D+      D3492 D3496 D3500  ; QTY數量
1599  LD=     K0 D10600
      AND=    K0 D10601
      AND=    K0 D10602
      AND=    K0 D10603
      AND=    K0 D10604
      AND=    K0 D10605
      AND=    K0 D10606
      AND=    K0 D10607
      AND=    K0 D10608
      AND=    K0 D10609
      INV
      OUT     M5900  ; SECS_上位下指令不為空
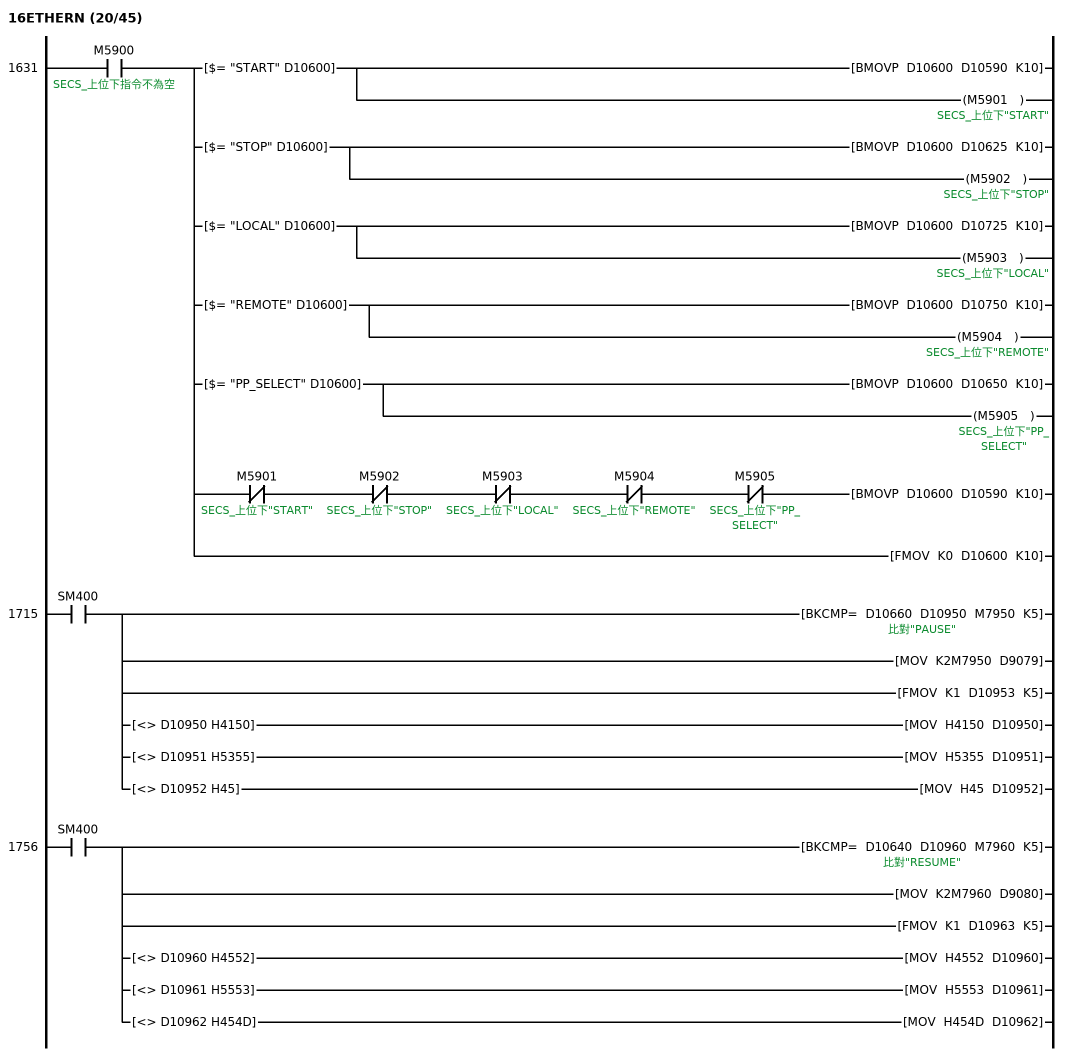
1631  LD      M5900  ; SECS_上位下指令不為空
      MPS
      AND$=   "START" D10600
      BMOVP   D10600 D10590 K10
      OUT     M5901  ; SECS_上位下"START"
      MRD
      AND$=   "STOP" D10600
      BMOVP   D10600 D10625 K10
      OUT     M5902  ; SECS_上位下"STOP"
      MRD
      AND$=   "LOCAL" D10600
      BMOVP   D10600 D10725 K10
      OUT     M5903  ; SECS_上位下"LOCAL"
      MRD
      AND$=   "REMOTE" D10600
      BMOVP   D10600 D10750 K10
      OUT     M5904  ; SECS_上位下"REMOTE"
      MRD
      AND$=   "PP_SELECT" D10600
      BMOVP   D10600 D10650 K10
      OUT     M5905  ; SECS_上位下"PP_SELECT"
      MRD
      ANI     M5901  ; SECS_上位下"START"
      ANI     M5902  ; SECS_上位下"STOP"
      ANI     M5903  ; SECS_上位下"LOCAL"
      ANI     M5904  ; SECS_上位下"REMOTE"
      ANI     M5905  ; SECS_上位下"PP_SELECT"
      BMOVP   D10600 D10590 K10
      MPP
      FMOV    K0 D10600 K10
1715  LD      SM400
      BKCMP=  D10660 D10950 M7950 K5  ; 比對"PAUSE"
        [note] 上位下PAUSE指令
      MOV     K2M7950 D9079
      FMOV    K1 D10953 K5
      MPS
      AND<>   D10950 H4150
      MOV     H4150 D10950
      MRD
      AND<>   D10951 H5355
      MOV     H5355 D10951
      MPP
      AND<>   D10952 H45
      MOV     H45 D10952
1756  LD      SM400
      BKCMP=  D10640 D10960 M7960 K5  ; 比對"RESUME"
        [note] 上位下RESUME指令
      MOV     K2M7960 D9080
      FMOV    K1 D10963 K5
      MPS
      AND<>   D10960 H4552
      MOV     H4552 D10960
      MRD
      AND<>   D10961 H5553
      MOV     H5553 D10961
      MPP
      AND<>   D10962 H454D
      MOV     H454D D10962
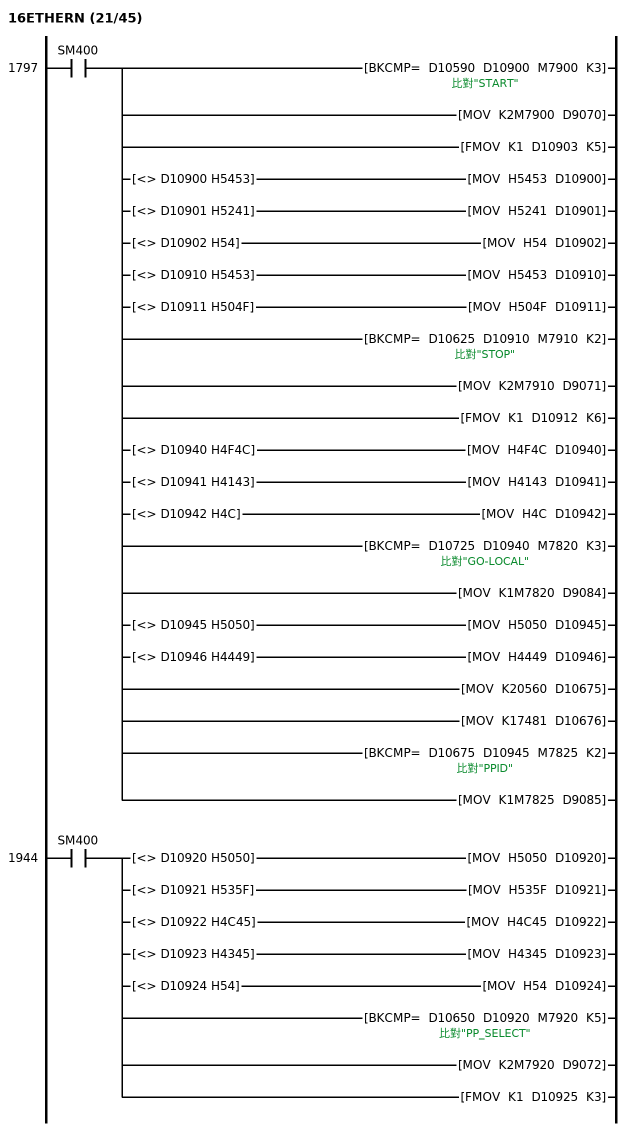
1797  LD      SM400
      BKCMP=  D10590 D10900 M7900 K3  ; 比對"START"
        [note] 上位下START指令
      MOV     K2M7900 D9070
      FMOV    K1 D10903 K5
      MPS
      AND<>   D10900 H5453
      MOV     H5453 D10900
      MRD
      AND<>   D10901 H5241
      MOV     H5241 D10901
      MRD
      AND<>   D10902 H54
      MOV     H54 D10902
      MRD
      AND<>   D10910 H5453
      MOV     H5453 D10910
      MRD
      AND<>   D10911 H504F
      MOV     H504F D10911
      MPP
      BKCMP=  D10625 D10910 M7910 K2  ; 比對"STOP"
        [note] 上位下STOP指令
      MOV     K2M7910 D9071
      FMOV    K1 D10912 K6
      MPS
      AND<>   D10940 H4F4C
      MOV     H4F4C D10940
      MRD
      AND<>   D10941 H4143
      MOV     H4143 D10941
      MRD
      AND<>   D10942 H4C
      MOV     H4C D10942
      MPP
      BKCMP=  D10725 D10940 M7820 K3  ; 比對"GO-LOCAL"
        [note] 上位下GO-LOCAL指令
      MOV     K1M7820 D9084
      MPS
      AND<>   D10945 H5050
      MOV     H5050 D10945
      MRD
      AND<>   D10946 H4449
      MOV     H4449 D10946
      MPP
      MOV     K20560 D10675
      MOV     K17481 D10676
      BKCMP=  D10675 D10945 M7825 K2  ; 比對"PPID"
        [note] 上位下PPID指令
      MOV     K1M7825 D9085
1944  LD      SM400
      MPS
      AND<>   D10920 H5050
      MOV     H5050 D10920
      MRD
      AND<>   D10921 H535F
      MOV     H535F D10921
      MRD
      AND<>   D10922 H4C45
      MOV     H4C45 D10922
      MRD
      AND<>   D10923 H4345
      MOV     H4345 D10923
      MRD
      AND<>   D10924 H54
      MOV     H54 D10924
      MPP
      BKCMP=  D10650 D10920 M7920 K5  ; 比對"PP_SELECT"
        [note] 上位下PP_SELECT指令
      MOV     K2M7920 D9072
      FMOV    K1 D10925 K3
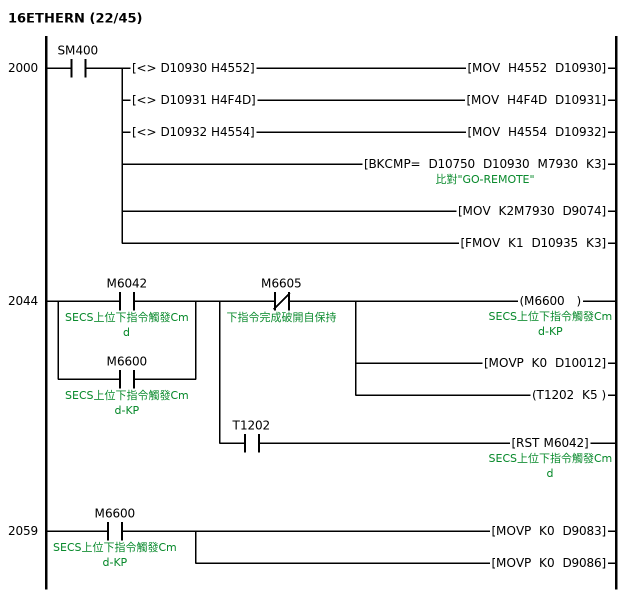
2000  LD      SM400
      MPS
      AND<>   D10930 H4552
      MOV     H4552 D10930
      MRD
      AND<>   D10931 H4F4D
      MOV     H4F4D D10931
      MRD
      AND<>   D10932 H4554
      MOV     H4554 D10932
      MPP
      BKCMP=  D10750 D10930 M7930 K3  ; 比對"GO-REMOTE"
        [note] 上位下GO-REMOTE指令
      MOV     K2M7930 D9074
      FMOV    K1 D10935 K3
2044  LD      M6042  ; SECS上位下指令觸發Cmd
      OR      M6600  ; SECS上位下指令觸發Cmd-KP
      MPS
      ANI     M6605  ; 下指令完成破開自保持
      OUT     M6600  ; SECS上位下指令觸發Cmd-KP
      MOVP    K0 D10012
      OUT     T1202 K5
      MPP
      AND     T1202
      RST     M6042  ; SECS上位下指令觸發Cmd
2059  LD      M6600  ; SECS上位下指令觸發Cmd-KP
      MOVP    K0 D9083
      MOVP    K0 D9086
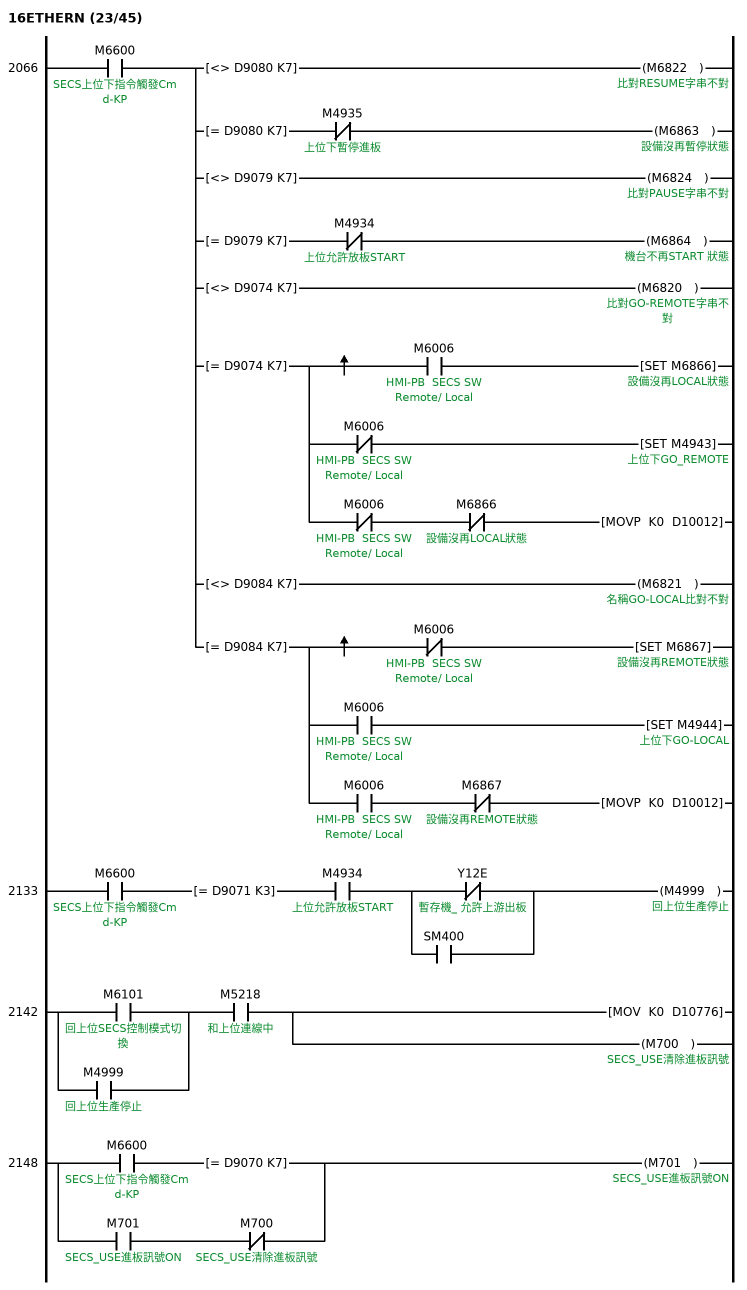
2066  LD      M6600  ; SECS上位下指令觸發Cmd-KP
      MPS
      AND<>   D9080 K7
      OUT     M6822  ; 比對RESUME字串不對
      MRD
      AND=    D9080 K7
      ANI     M4935  ; 上位下暫停進板
      OUT     M6863  ; 設備沒再暫停狀態
      MRD
      AND<>   D9079 K7
      OUT     M6824  ; 比對PAUSE字串不對
      MRD
      AND=    D9079 K7
      ANI     M4934  ; 上位允許放板START
      OUT     M6864  ; 機台不再START 狀態
      MRD
      AND<>   D9074 K7
      OUT     M6820  ; 比對GO-REMOTE字串不對
      MRD
      AND=    D9074 K7
      MPS
      MEP
      AND     M6006  ; HMI-PB  SECS SW  Remote/ Local
      SET     M6866  ; 設備沒再LOCAL狀態
      MRD
      ANI     M6006  ; HMI-PB  SECS SW  Remote/ Local
      SET     M4943  ; 上位下GO_REMOTE
      MPP
      ANI     M6006  ; HMI-PB  SECS SW  Remote/ Local
      ANI     M6866  ; 設備沒再LOCAL狀態
      MOVP    K0 D10012
      MRD
      AND<>   D9084 K7
      OUT     M6821  ; 名稱GO-LOCAL比對不對
      MPP
      AND=    D9084 K7
      MPS
      MEP
      ANI     M6006  ; HMI-PB  SECS SW  Remote/ Local
      SET     M6867  ; 設備沒再REMOTE狀態
      MRD
      AND     M6006  ; HMI-PB  SECS SW  Remote/ Local
      SET     M4944  ; 上位下GO-LOCAL
      MPP
      AND     M6006  ; HMI-PB  SECS SW  Remote/ Local
      ANI     M6867  ; 設備沒再REMOTE狀態
      MOVP    K0 D10012
2133  LD      M6600  ; SECS上位下指令觸發Cmd-KP
      AND=    D9071 K3
      AND     M4934  ; 上位允許放板START
      LDI     Y12E  ; 暫存機_ 允許上游出板
      OR      SM400
      ANB
      OUT     M4999  ; 回上位生產停止
2142  LD      M6101  ; 回上位SECS控制模式切換
      OR      M4999  ; 回上位生產停止
      AND     M5218  ; 和上位連線中
      MOV     K0 D10776
      OUT     M700  ; SECS_USE清除進板訊號
2148  LD      M6600  ; SECS上位下指令觸發Cmd-KP
      AND=    D9070 K7
      LD      M701  ; SECS_USE進板訊號ON
      ANI     M700  ; SECS_USE清除進板訊號
      ORB
      OUT     M701  ; SECS_USE進板訊號ON
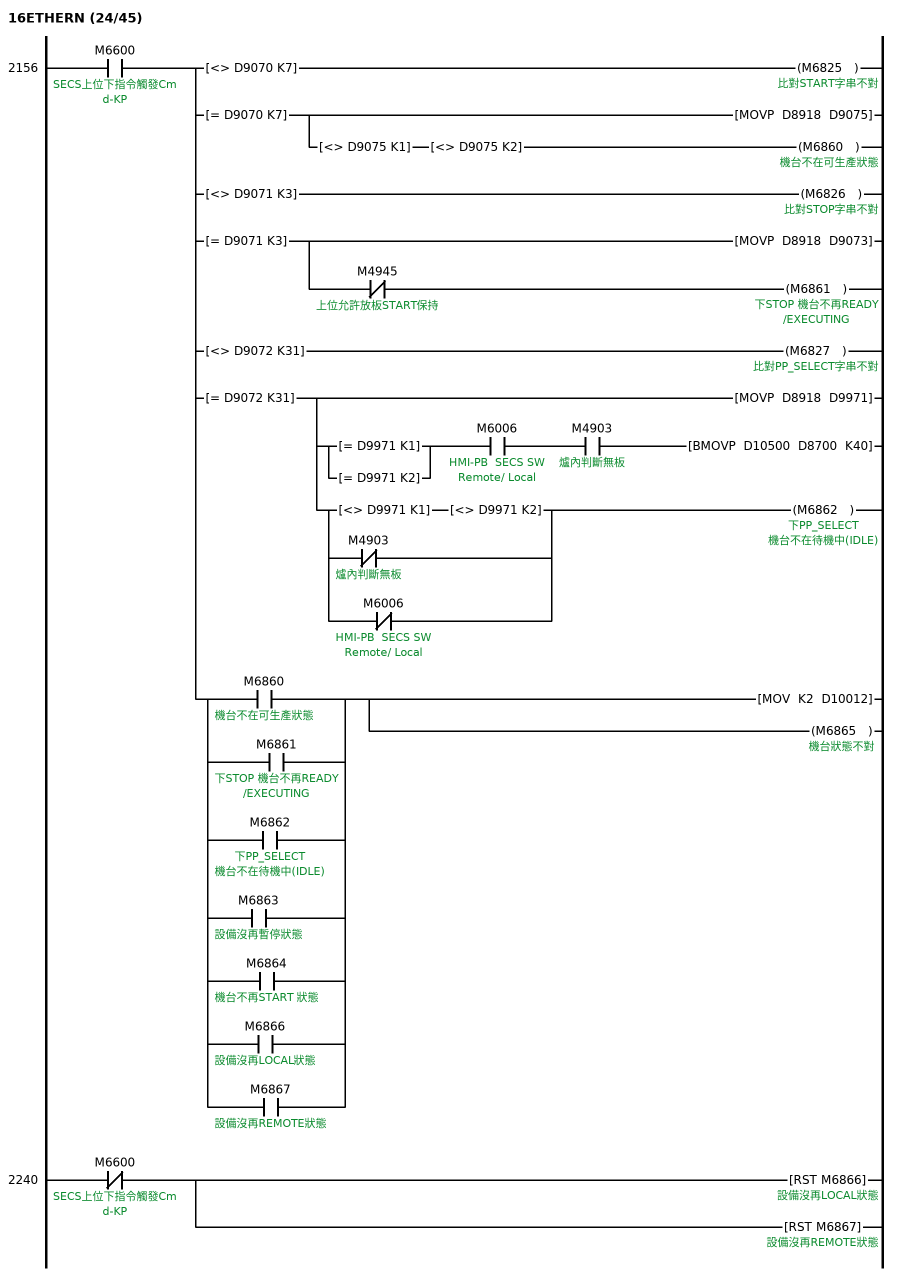
2156  LD      M6600  ; SECS上位下指令觸發Cmd-KP
      MPS
      AND<>   D9070 K7
      OUT     M6825  ; 比對START字串不對
      MRD
      AND=    D9070 K7
      MOVP    D8918 D9075
      AND<>   D9075 K1
      AND<>   D9075 K2
      OUT     M6860  ; 機台不在可生產狀態
      MRD
      AND<>   D9071 K3
      OUT     M6826  ; 比對STOP字串不對
      MRD
      AND=    D9071 K3
      MOVP    D8918 D9073
      ANI     M4945  ; 上位允許放板START保持
      OUT     M6861  ; 下STOP 機台不再READY/EXECUTING
      MRD
      AND<>   D9072 K31
      OUT     M6827  ; 比對PP_SELECT字串不對
      MRD
      AND=    D9072 K31
      MOVP    D8918 D9971
      MPS
      LD=     D9971 K1
      OR=     D9971 K2
      ANB
      AND     M6006  ; HMI-PB  SECS SW  Remote/ Local
      AND     M4903  ; 爐內判斷無板
      BMOVP   D10500 D8700 K40
      MPP
      LD<>    D9971 K1
      AND<>   D9971 K2
      ORI     M4903  ; 爐內判斷無板
      ORI     M6006  ; HMI-PB  SECS SW  Remote/ Local
      ANB
      OUT     M6862  ; 下PP_SELECT 機台不在待機中(IDLE)
      MPP
      LD      M6860  ; 機台不在可生產狀態
      OR      M6861  ; 下STOP 機台不再READY/EXECUTING
      OR      M6862  ; 下PP_SELECT 機台不在待機中(IDLE)
      OR      M6863  ; 設備沒再暫停狀態
      OR      M6864  ; 機台不再START 狀態
      OR      M6866  ; 設備沒再LOCAL狀態
      OR      M6867  ; 設備沒再REMOTE狀態
      ANB
      MOV     K2 D10012
      OUT     M6865  ; 機台狀態不對
2240  LDI     M6600  ; SECS上位下指令觸發Cmd-KP
      RST     M6866  ; 設備沒再LOCAL狀態
      RST     M6867  ; 設備沒再REMOTE狀態
